# B&R Automation Studio project awecoRT
Automation Studio 4.2.7.54 SP

## Configuration Config1

CPU X20CP1381, AutomationRuntime A4.26, Build 4.1.2, Vc V4.26.1

### Task classes (Cpu.sw)
```
Cyclic#1 (cycle 2000 us, tolerance 0 us):
  SinSignal <- SinSignal.prg
Binaries: TCData, arconfig, asfw, ashwd, iomap, User, Role, sysconf
ReActionTechnologyObjects: Program <- Program.prg
Libraries: AsIORTI, astime, asieccon, runtime
```

### Hardware
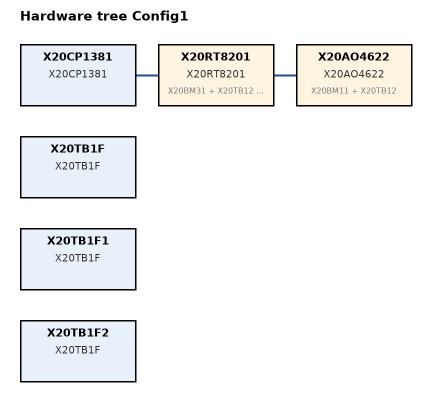
```
X20AO4622 : X20AO4622 v1.0.6.1  [SS1 -> X20TB12b.SS; SL -> X20BM11.SL1]
X20BM11 : X20BM11 v1.0.0.1  [X2X1 -> X20BM31.X2X2]
X20BM31 : X20BM31 v1.0.0.1  [X2X1 -> X20CP1381.IF6]
X20CP1381 : X20CP1381 v1.3.2.0  [X1 -> X1.SL; X2 -> X2.SL; X3 -> X3.SL]
  Module X1 (Type=X1, Virtual=true, Version=1.0.0.0)
    Connection (Connector=SS1, TargetModule=X20TB1F, TargetConnector=SS)
    Connection (Connector=SL, TargetModule=X20CP1381, TargetConnector=X1)
  Module X2 (Type=X2, Virtual=true, Version=1.0.0.0)
    Connection (Connector=SS1, TargetModule=X20TB1F1, TargetConnector=SS)
    Connection (Connector=SL, TargetModule=X20CP1381, TargetConnector=X2)
  Module X3 (Type=X3, Virtual=true, Version=1.0.0.0)
    Connection (Connector=SS1, TargetModule=X20TB1F2, TargetConnector=SS)
    Connection (Connector=SL, TargetModule=X20CP1381, TargetConnector=X3)
  Connector IF2:
    ActivateDevice = 1
    Mode = Manual
    InternetAddress = 192.168.0.105
    SubnetMask = 255.255.255.0
  ConfigurationID = rt8201_Config1
  TimerDeviceType = SWIOTIMER
  SystemTick = 2000
  Cyclic1Duration = 2000
  Cyclic1Tolerance = 0
  Cyclic2Duration = 20000
  Cyclic2Tolerance = 20000
  Cyclic3Duration = 50000
  Cyclic3Tolerance = 50000
  Cyclic4Duration = 100000
  Cyclic4Tolerance = 100000
  Cyclic5Duration = 200000
  Cyclic5Tolerance = 200000
  Cyclic6Duration = 500000
  Cyclic6Tolerance = 500000
  Cyclic7Duration = 1000000
  Cyclic7Tolerance = 1000000
  Cyclic8Duration = 10000
  Cyclic8Tolerance = 30000000
X20RT8201 : X20RT8201 v1.1.0.0  [SS1 -> X20TB12.SS; SS2 -> X20TB12a.SS; SL -> X20BM31.SL1]
  ReActionTask = Program
  ReActionTaskDisabled = FALSE
  ReActionCycleTime = 1
  ReActionCycleCounter = on
  ReActionCycleTimeMin = on
  TypeRes1 = DINT
  TypeRes2 = BOOL
X20TB12 : X20TB12 v1.0.0.0
X20TB12a : X20TB12 v1.0.0.0
X20TB12b : X20TB12 v1.0.0.0
X20TB1F : X20TB1F v1.0.0.0
X20TB1F1 : X20TB1F v1.0.0.0
X20TB1F2 : X20TB1F v1.0.0.0
```

### IoMap.iom - X20CP1381/IoMap.iom
```iecst
VAR_CONFIG
	::SinSignal:RTCycleCounter AT %IW."X20RT8201".RTCycleCounter;
	::SinSignal:di1 AT %IX."X1".DigitalInput01;
	::SinSignal:RTEnable AT %QX."X20RT8201".RTEnable;
	::SinSignal:sin_val AT %QW."X20AO4622".AnalogOutput01;
END_VAR
```

## Configuration X20CP1584

CPU X20CP1584, AutomationRuntime A4.26, Build 4.1.2, Vc V4.26.2

### Task classes (Cpu.sw)
```
Cyclic#1 (cycle 500 us, tolerance 0 us):
  TyrControl <- TyrControl.prg
Cyclic#2 (cycle 1000 us, tolerance 0 us):
  SinSignal <- SinSignal.prg
Binaries: TCData, arconfig, asfw, ashwd, iomap, User, Role, sysconf
ReActionTechnologyObjects: Program <- Program.prg
Libraries: astime, asieccon, sys_lib, AsBrStr, runtime, asiorti
```

### Hardware
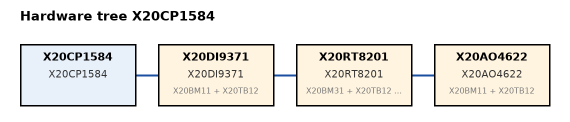
```
X20AO4622 : X20AO4622 v1.0.6.1  [SS1 -> X20TB12c.SS; SL -> X20BM11a.SL1]
X20BM11 : X20BM11 v1.0.0.1  [X2X1 -> X20CP1584.IF6]
X20BM11a : X20BM11 v1.0.0.1  [X2X1 -> X20BM31.X2X2]
X20BM31 : X20BM31 v1.0.0.1  [X2X1 -> X20BM11.X2X2]
X20CP1584 : X20CP1584 v1.3.0.0
  Connector IF2:
    ActivateDevice = 1
    EthInterfaceRedundant = 0
  Connector IF3:
    EplInterfaceRedundant = 0
    EplEthInterfaceRedundant = 0
  Connector IF6:
    CycleTime = 500
  ConfigurationID = rt8201_X20CP1584
  TimerDeviceType = SWIOTIMER
  SystemTick = 500
  IdleTaskClass = 3
  Cyclic1Duration = 500
  Cyclic1Tolerance = 0
  Cyclic2Duration = 1000
  Cyclic2Tolerance = 0
  Cyclic3Duration = 50000
  Cyclic3Tolerance = 50000
  Cyclic4Duration = 100000
  Cyclic4Tolerance = 100000
  Cyclic5Duration = 200000
  Cyclic5Tolerance = 200000
  Cyclic6Duration = 500000
  Cyclic6Tolerance = 500000
  Cyclic7Duration = 1000000
  Cyclic7Tolerance = 1000000
  Cyclic8Duration = 10000
  Cyclic8Tolerance = 30000000
X20DI9371 : X20DI9371 v1.0.1.3  [SS1 -> X20TB12.SS; SL -> X20BM11.SL1]
  InputFilter = 0
X20RT8201 : X20RT8201 v1.1.0.0  [SS1 -> X20TB12a.SS; SS2 -> X20TB12b.SS; SL -> X20BM31.SL1]
  ReActionTask = Program
  ReActionTaskDisabled = FALSE
  ReActionCycleTime = 1
  ReActionCycleCounter = on
  ReActionCycleTimeMin = on
  TypePar1 = DINT
  TypeRes1 = BOOL
X20TB12 : X20TB12 v1.0.0.0
X20TB12a : X20TB12 v1.0.0.0
X20TB12b : X20TB12 v1.0.0.0
X20TB12c : X20TB12 v1.0.0.0
```

### IoMap.iom - X20CP1584/IoMap.iom
```iecst
VAR_CONFIG
	::SinSignal:RTEnable AT %QX."X20RT8201".RTEnable;
	Cyclic#1.::di1 AT %IX."X20DI9371".DigitalInput01;
	Cyclic#1.::sin_val AT %QW."X20AO4622".AnalogOutput01;
	Cyclic#1.::TyrControl:analogOutput02 AT %QW."X20AO4622".AnalogOutput02;
	Cyclic#1.::Par1 AT %QD."X20RT8201".PAR01;
	Cyclic#1.::RES01Bit1 AT %IX."X20RT8201".RES01_Bit1;
	Cyclic#1.::RES01Bit2 AT %IX."X20RT8201".RES01_Bit2;
	Cyclic#1.::RES01Bit3  AT %IX."X20RT8201".RES01_Bit3;
END_VAR
```

## Logical view

Binary libraries used (declarations not repeated): operator, runtime, astime, AsIecCon, AsIORTI, sys_lib, AsBrStr

### Global.var - Global variables
```iecst
VAR
	di1 : BOOL;
	sin_val : INT;
	Par1 : DINT;
	RES01Bit1 : BOOL;
	RES01Bit2 : BOOL;
	RES01Bit3 : BOOL;
END_VAR
```


### Program Logical/Program (ReAction)

#### Variables.var
```iecst
VAR
	rtiAin_0 : rtiAin;
	rtiRes_0 : rtiRes;
	rtiComp_0 : rtiComp;
	rtiRes_1 : rtiRes;
	rtiAnLimit_0 : rtiAnLimit;
	rtiDout_0 : rtiDout;
	rtiTP_0 : rtiTP;
	rtiPar_0 : rtiPar;
	rtiComp_1 : rtiComp;
	rtiRes_2 : rtiRes;
	rtiNot_0 : rtiNot;
	rtiTP_1 : rtiTP;
	rtiDout_1 : rtiDout;
	rtiRes_3 : rtiRes;
	rtiXor_0 : rtiXor;
	rtiOr_0 : rtiOr;
	rtiXor_1 : rtiXor;
	rtiOr_1 : rtiOr;
END_VAR
```

- Cyclic.rti (not shown)

### Program Logical/SinSignal (IEC)

#### Cyclic.st - Cyclic code
```iecst
PROGRAM _INIT

	RTCycleCounter;
	RTEnable := TRUE;
	edgeCase := 0;
END_PROGRAM

PROGRAM _CYCLIC

	CASE edgeCase OF
		RISE:
			alpha_rad := ((PI/10)*tmp);
			IF tmp = 5 THEN
				tmp := 4;
				edgeCase := FALL;
			ELSE
				tmp := tmp +1;
			END_IF;
		FALL:
			alpha_rad := ((PI/10)*tmp);
			IF tmp = -5 THEN
				tmp := -4;
				edgeCase := RISE;
			ELSE
				tmp := tmp - 1;
			END_IF;
	END_CASE;

	sin_val := REAL_TO_INT(32000*SIN(alpha_rad));

	di1;

	RES01Bit1;
	RES01Bit2;

END_PROGRAM
```

#### Types.typ - Local data types
```iecst
TYPE
	edge_type :
		(
		RISE := 0,
		FALL := 1
		);
END_TYPE
```

#### Variables.var - Local variables
```iecst
VAR CONSTANT
	PI : REAL := 3.1415926535897932384626433832795;
	k : REAL := 3.1830988618379067153776752674503;
END_VAR
VAR
	edgeCase : edge_type;
	tmp : INT;
	RTEnable : BOOL;
	RTCycleCounter : UINT;
	alpha_rad : REAL;
END_VAR
```

### Program Logical/TyrControl (IEC)

#### Main.st - Init, cyclic, exit code
```iecst
PROGRAM _INIT
	(* Insert code here *)
	DimmerPow := 40;
	Par1 := 5000;
END_PROGRAM

PROGRAM _CYCLIC
	Par1;
(*	DimmerTime := REAL_TO_INT(DimmerPow * 0.18);

	CASE BOOL_TO_INT(RES02Bit1) OF
		0:
			tmp2 := 0;
			IF tmp1 < DimmerTime THEN
				analogOutput02 := DINT_TO_INT(RES01);
			ELSE
				analogOutput02 := 0;
			END_IF;
		tmp1 := tmp1 +1;

		1:
			tmp1 := 0;
			IF tmp2 < DimmerTime THEN
				analogOutput02 := DINT_TO_INT(RES01);
			ELSE
				analogOutput02 := 0;
			END_IF;
		tmp2 := tmp2 +1;
	END_CASE;
*)
END_PROGRAM
```

#### Variables.var - Local variables
```iecst
VAR
	DimmerTime : UINT;
	DimmerPow : REAL;
	tmp1 : UINT;
	analogOutput02 : INT;
	tmp2 : UINT;
END_VAR
```

Listed in the project but not available here: Logical/Global.typ, Logical/TyrControl/Types.typ
